FUNCTION_BLOCK FB_SaveasCSVFile IMPLEMENTS I_PersistentEventStorage
VAR_INPUT
END_VAR
VAR_OUTPUT
END_VAR
VAR
	fileopen : FB_FileOpen:= (sPathName:= 'C:\Users\ramak\Downloads\Event Logger\Events.log',nMode:= FOPEN_MODEAPPEND OR FOPEN_MODETEXT);
	fileputs :  FB_FilePuts;
	eWriteState : (fileOpenTrigger, fileOpen, waitForTheEvent,eventWriteTrigger, eventWrite, fileClose, errorHandeling);
	stEventWriteToFile : ST_Event;
	createdCSVString : T_MaxString;
	fbEventRingBuffer : FB_EventRingBuffer;
END_VAR

CASE eWriteState OF
	fileOpenTrigger: 
		fileopen(bExecute:= TRUE);
		eWriteState := fileOpen;
		
	fileOpen :
		fileopen(bExecute:= FALSE);
		IF fileopen.bError THEN
			eWriteState:= errorHandeling;
		ELSIF NOT fileopen.bBusy AND fileopen.hFile <> 0 THEN
			eWriteState := waitForTheEvent;
		END_IF
	waitForTheEvent :
		    IF fbEventRingBuffer.Remove(stEvent => stEventWriteToFile) THEN
        eWriteState := eventWriteTrigger;
    END_IF

	eventWriteTrigger :
		createdCSVString := concatString(stEvent:= stEventWriteToFile);
		fileputs(bExecute:= TRUE, sLine:=createdCSVString, hFile:=fileopen.hFile);
		eWriteState:= eventWrite;
		
	eventWrite:
		fileputs(bExecute:= FALSE);
		IF fileputs.bError THEN
			eWriteState:= errorHandeling;
			ELSIF NOT fileputs.bBusy THEN
				eWriteState:= waitForTheEvent;
		END_IF
		
	errorHandeling :
	//noting
	
END_CASE

METHOD PRIVATE concatString : T_MaxString
VAR_INPUT
	stEvent : REFERENCE TO ST_Event;
END_VAR
VAR
	stringFlag : T_MaxString;
END_VAR
stringFlag:= TO_STRING(stEvent.eEventType);
stringFlag := CONCAT(STR1:= stringFlag, STR2:= TO_STRING(stEvent.eEventSeverity));
stringFlag := CONCAT(STR1:= stringFlag, STR2:= ',');
stringFlag := CONCAT(STR1:= stringFlag, STR2:= TO_STRING(stEvent.dtTimeStamp));
stringFlag := CONCAT(STR1:= stringFlag, STR2:= ',');
stringFlag := CONCAT(STR1:= stringFlag, STR2:= TO_STRING(stEvent.nEventIdentity));
stringFlag := CONCAT(STR1:= stringFlag, STR2:= ',');
stringFlag := CONCAT(STR1:= stringFlag, STR2:= stEvent.sEventText);
stringFlag := CONCAT(STR1:= stringFlag, STR2:= '\n');
concatString := stringFlag;
END_METHOD

METHOD storeEvent
VAR_INPUT
	stEvent	: ST_Event;
END_VAR
VAR
	fbEventRingBuffer : FB_EventRingBuffer;
END_VAR
fbEventRingBuffer.Apend(stEvent:=stEvent);


//IF eWriteState = waitForTheEvent THEN
	//eWriteState := eventWriteTrigger;
	//stEventWriteToFile :=stEvent;
//END_IF
END_METHOD

END_FUNCTION_BLOCK

(* stored: Version 1.1.0.1, ProductVersion 3.1.4024.16
   POU FB_SaveasCSVFile: Id {01ae8648-2ac2-4edc-95e4-525f41831fd8}, SpecialFunc None
   Method concatString: Id {327be36b-a4dc-4aeb-94e1-1dacfd82036f}
   Method storeEvent: Id {c392af54-cbd9-408d-9f08-46672b69169e} *)
